VISUALIZATION visutest  // 2x2
END_VISUALIZATION

(* stored: Version 1.1.0.1, ProductVersion 3.1.4020.12
   Visu visutest: Id {5bef4dce-a1fe-48f7-bc87-09637add1255} *)
